PROGRAM PRG_PLAS_18_InterimCamCtrl
VAR

	bEnableInterimCameraSystem 	: BOOL;

	tofInterimCameraOFFDelay 		: TOF;

	fbInterimShiftQueue				: FB_PLAS_InterimShiftQueue;
	fbInterimCamera		: FB_SCANNER_CameraSelect;
	fbInterimEvaluation		: FB_SCANNER_Evaluation;

	rtrigNewArrived					: R_TRIG;
	bNewCodeIsProccesing			: BOOL;

	tonValidationTimout				: TON;
	bValidationTimeout				: BOOL;
	bValidationTimeoutReset			: BOOL;

	fbAddInterimCodeToQ				: FB_PLAS_AddInterimCodeToQ;
	rtrigDuplicateDetection			: R_TRIG;

	fbDebugCNT						: FB_DEBUG_CounterArray;
	aCNTDebug						: ARRAY [1..10] OF UDINT;
	bResetCNT							: BOOL;

END_VAR

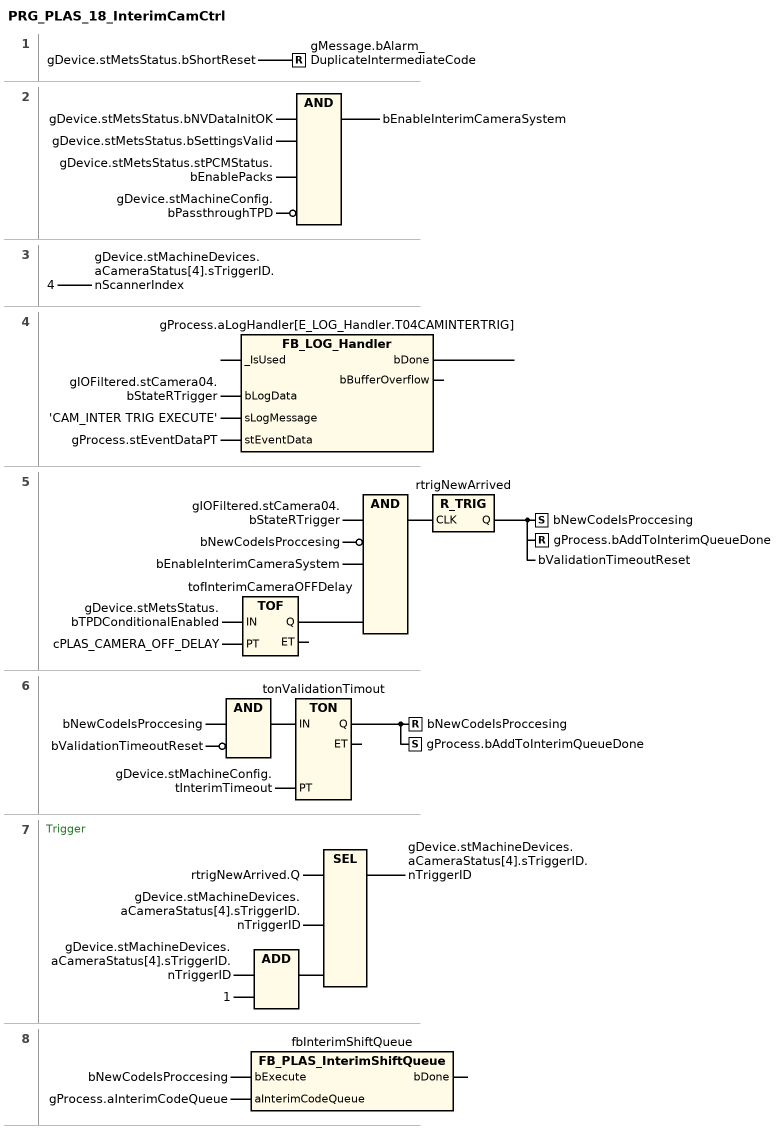
// NETWORK 1
gMessage.bAlarm_DuplicateIntermediateCode R= gDevice.stMetsStatus.bShortReset;

// NETWORK 2
bEnableInterimCameraSystem := gDevice.stMetsStatus.bNVDataInitOK AND gDevice.stMetsStatus.bSettingsValid AND gDevice.stMetsStatus.stPCMStatus.bEnablePacks AND NOT gDevice.stMachineConfig.bPassthroughTPD;

// NETWORK 3
gDevice.stMachineDevices.aCameraStatus[4].sTriggerID.nScannerIndex := 4;

// NETWORK 4
gProcess.aLogHandler[E_LOG_Handler.T04CAMINTERTRIG](
    bLogData := gIOFiltered.stCamera04.bStateRTrigger,
    sLogMessage := 'CAM_INTER TRIG EXECUTE',
    stEventData := gProcess.stEventDataPT); // FB_LOG_Handler

// NETWORK 5
tofInterimCameraOFFDelay(IN := gDevice.stMetsStatus.bTPDConditionalEnabled, PT := cPLAS_CAMERA_OFF_DELAY); // TOF
rtrigNewArrived(CLK := gIOFiltered.stCamera04.bStateRTrigger AND NOT bNewCodeIsProccesing AND bEnableInterimCameraSystem AND tofInterimCameraOFFDelay.Q); // R_TRIG
bNewCodeIsProccesing S= rtrigNewArrived.Q;
gProcess.bAddToInterimQueueDone R= rtrigNewArrived.Q;
bValidationTimeoutReset := rtrigNewArrived.Q;

// NETWORK 6
tonValidationTimout(IN := bNewCodeIsProccesing AND NOT bValidationTimeoutReset, PT := gDevice.stMachineConfig.tInterimTimeout); // TON
bNewCodeIsProccesing R= tonValidationTimout.Q;
gProcess.bAddToInterimQueueDone S= tonValidationTimout.Q;

// NETWORK 7
// Trigger
gDevice.stMachineDevices.aCameraStatus[4].sTriggerID.nTriggerID := SEL(rtrigNewArrived.Q, gDevice.stMachineDevices.aCameraStatus[4].sTriggerID.nTriggerID, gDevice.stMachineDevices.aCameraStatus[4].sTriggerID.nTriggerID + 1);

// NETWORK 8
fbInterimShiftQueue(bExecute := bNewCodeIsProccesing, aInterimCodeQueue := gProcess.aInterimCodeQueue); // FB_PLAS_InterimShiftQueue

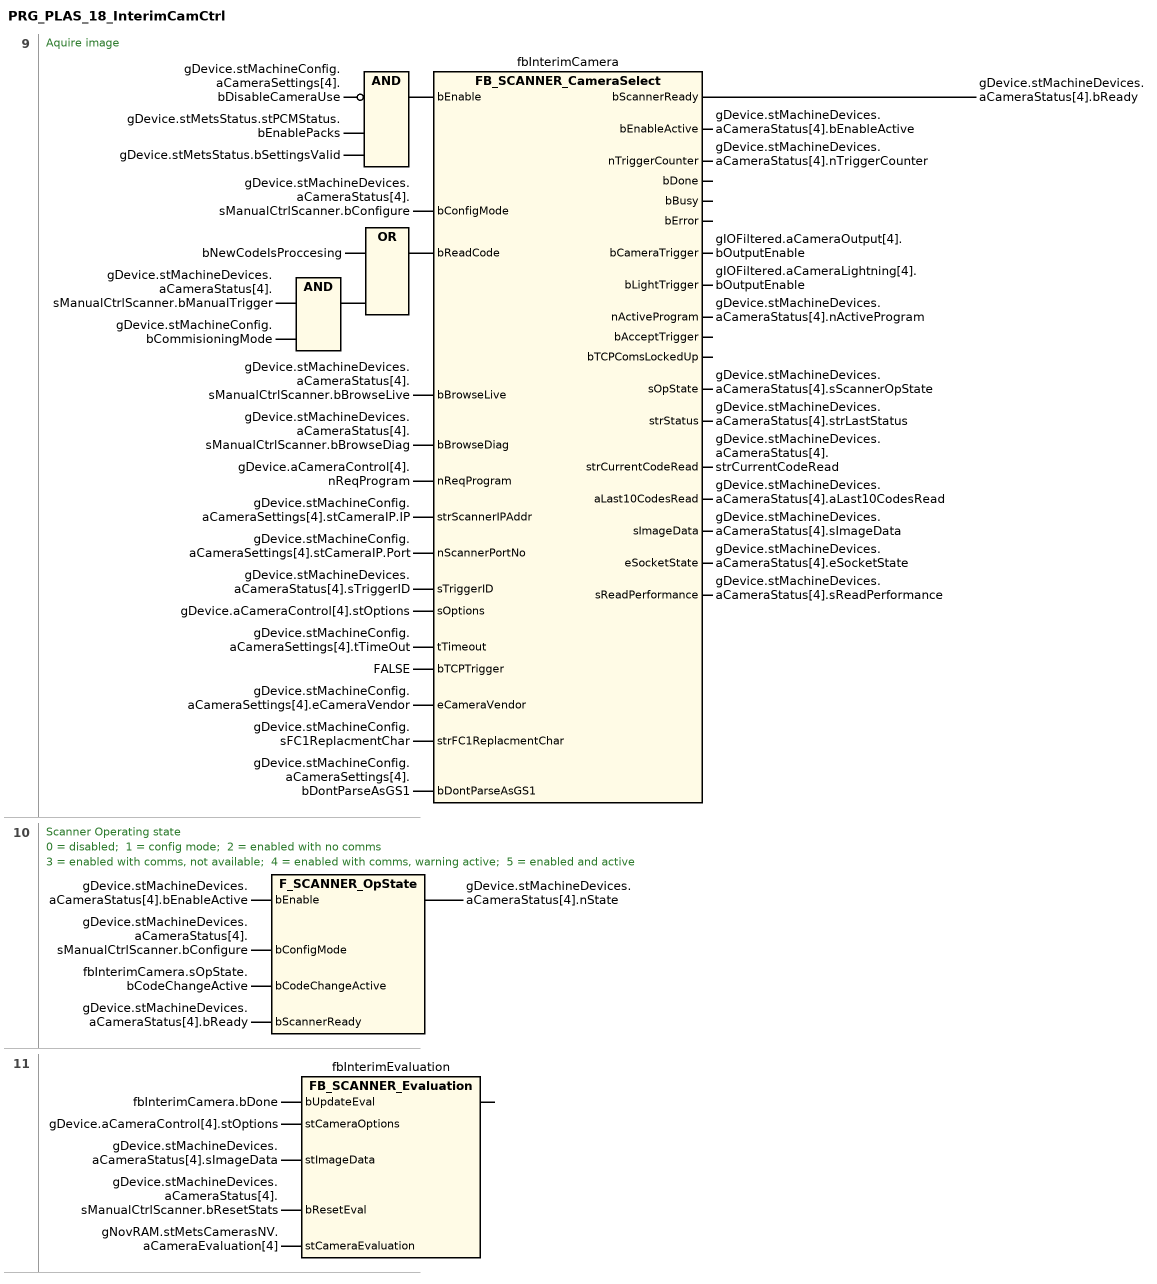
// NETWORK 9
// Aquire image
fbInterimCamera(
    bEnable := NOT gDevice.stMachineConfig.aCameraSettings[4].bDisableCameraUse AND gDevice.stMetsStatus.stPCMStatus.bEnablePacks AND gDevice.stMetsStatus.bSettingsValid,
    bConfigMode := gDevice.stMachineDevices.aCameraStatus[4].sManualCtrlScanner.bConfigure,
    bReadCode := bNewCodeIsProccesing OR gDevice.stMachineDevices.aCameraStatus[4].sManualCtrlScanner.bManualTrigger AND gDevice.stMachineConfig.bCommisioningMode,
    bBrowseLive := gDevice.stMachineDevices.aCameraStatus[4].sManualCtrlScanner.bBrowseLive,
    bBrowseDiag := gDevice.stMachineDevices.aCameraStatus[4].sManualCtrlScanner.bBrowseDiag,
    nReqProgram := gDevice.aCameraControl[4].nReqProgram,
    strScannerIPAddr := gDevice.stMachineConfig.aCameraSettings[4].stCameraIP.IP,
    nScannerPortNo := gDevice.stMachineConfig.aCameraSettings[4].stCameraIP.Port,
    sTriggerID := gDevice.stMachineDevices.aCameraStatus[4].sTriggerID,
    sOptions := gDevice.aCameraControl[4].stOptions,
    tTimeout := gDevice.stMachineConfig.aCameraSettings[4].tTimeOut,
    bTCPTrigger := FALSE,
    eCameraVendor := gDevice.stMachineConfig.aCameraSettings[4].eCameraVendor,
    strFC1ReplacmentChar := gDevice.stMachineConfig.sFC1ReplacmentChar,
    bDontParseAsGS1 := gDevice.stMachineConfig.aCameraSettings[4].bDontParseAsGS1,
    bEnableActive => gDevice.stMachineDevices.aCameraStatus[4].bEnableActive,
    nTriggerCounter => gDevice.stMachineDevices.aCameraStatus[4].nTriggerCounter,
    bCameraTrigger => gIOFiltered.aCameraOutput[4].bOutputEnable,
    bLightTrigger => gIOFiltered.aCameraLightning[4].bOutputEnable,
    nActiveProgram => gDevice.stMachineDevices.aCameraStatus[4].nActiveProgram,
    sOpState => gDevice.stMachineDevices.aCameraStatus[4].sScannerOpState,
    strStatus => gDevice.stMachineDevices.aCameraStatus[4].strLastStatus,
    strCurrentCodeRead => gDevice.stMachineDevices.aCameraStatus[4].strCurrentCodeRead,
    aLast10CodesRead => gDevice.stMachineDevices.aCameraStatus[4].aLast10CodesRead,
    sImageData => gDevice.stMachineDevices.aCameraStatus[4].sImageData,
    eSocketState => gDevice.stMachineDevices.aCameraStatus[4].eSocketState,
    sReadPerformance => gDevice.stMachineDevices.aCameraStatus[4].sReadPerformance); // FB_SCANNER_CameraSelect
gDevice.stMachineDevices.aCameraStatus[4].bReady := fbInterimCamera.bScannerReady;

// NETWORK 10
// 					Scanner Operating state
// 0 = disabled;  1 = config mode;  2 = enabled with no comms
// 3 = enabled with comms, not available;  4 = enabled with comms, warning active;  5 = enabled and active
//
gDevice.stMachineDevices.aCameraStatus[4].nState := F_SCANNER_OpState(bEnable := gDevice.stMachineDevices.aCameraStatus[4].bEnableActive, bConfigMode := gDevice.stMachineDevices.aCameraStatus[4].sManualCtrlScanner.bConfigure, bCodeChangeActive := fbInterimCamera.sOpState.bCodeChangeActive, bScannerReady := gDevice.stMachineDevices.aCameraStatus[4].bReady);

// NETWORK 11
fbInterimEvaluation(
    bUpdateEval := fbInterimCamera.bDone,
    stCameraOptions := gDevice.aCameraControl[4].stOptions,
    stImageData := gDevice.stMachineDevices.aCameraStatus[4].sImageData,
    bResetEval := gDevice.stMachineDevices.aCameraStatus[4].sManualCtrlScanner.bResetStats,
    stCameraEvaluation := gNovRAM.stMetsCamerasNV.aCameraEvaluation[4]); // FB_SCANNER_Evaluation

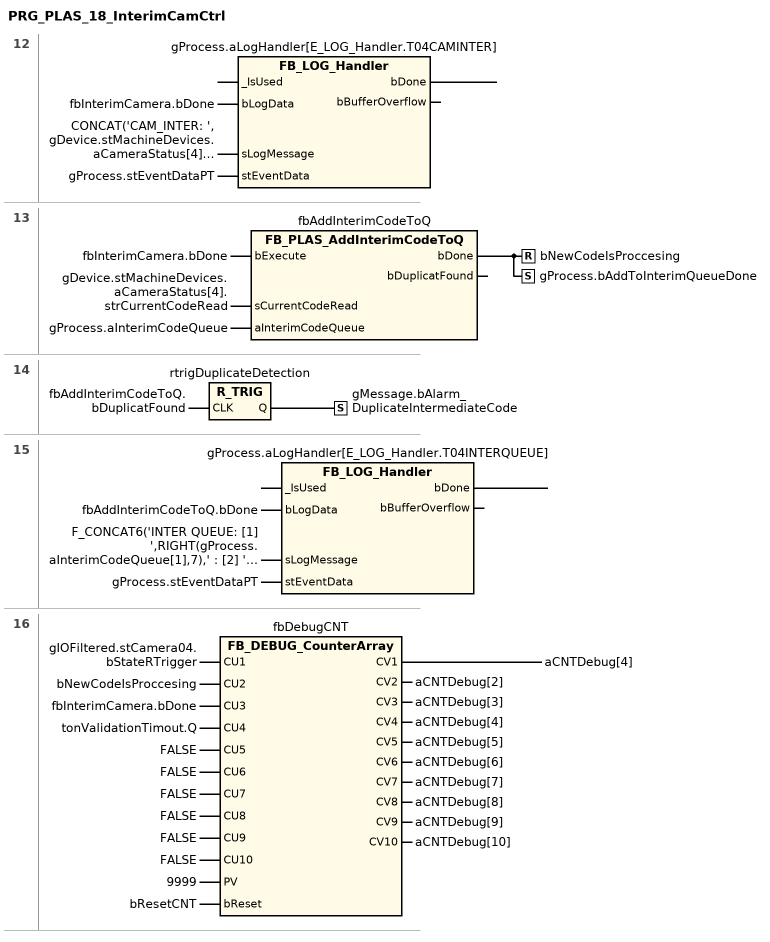
// NETWORK 12
gProcess.aLogHandler[E_LOG_Handler.T04CAMINTER](
    bLogData := fbInterimCamera.bDone,
    sLogMessage := CONCAT('CAM_INTER: ', gDevice.stMachineDevices.aCameraStatus[4].strCurrentCodeRead),
    stEventData := gProcess.stEventDataPT); // FB_LOG_Handler

// NETWORK 13
fbAddInterimCodeToQ(
    bExecute := fbInterimCamera.bDone,
    sCurrentCodeRead := gDevice.stMachineDevices.aCameraStatus[4].strCurrentCodeRead,
    aInterimCodeQueue := gProcess.aInterimCodeQueue); // FB_PLAS_AddInterimCodeToQ
bNewCodeIsProccesing R= fbAddInterimCodeToQ.bDone;
gProcess.bAddToInterimQueueDone S= fbAddInterimCodeToQ.bDone;

// NETWORK 14
rtrigDuplicateDetection(CLK := fbAddInterimCodeToQ.bDuplicatFound); // R_TRIG
gMessage.bAlarm_DuplicateIntermediateCode S= rtrigDuplicateDetection.Q;

// NETWORK 15
gProcess.aLogHandler[E_LOG_Handler.T04INTERQUEUE](
    bLogData := fbAddInterimCodeToQ.bDone,
    sLogMessage := F_CONCAT6('INTER QUEUE: [1] ',RIGHT(gProcess.aInterimCodeQueue[1],7),' : [2] ', RIGHT(gProcess.aInterimCodeQueue[2],7), ' : [3] ', RIGHT(gProcess.aInterimCodeQueue[3],7)),
    stEventData := gProcess.stEventDataPT); // FB_LOG_Handler

// NETWORK 16
fbDebugCNT(
    CU1 := gIOFiltered.stCamera04.bStateRTrigger,
    CU2 := bNewCodeIsProccesing,
    CU3 := fbInterimCamera.bDone,
    CU4 := tonValidationTimout.Q,
    CU5 := FALSE,
    CU6 := FALSE,
    CU7 := FALSE,
    CU8 := FALSE,
    CU9 := FALSE,
    CU10 := FALSE,
    PV := 9999,
    bReset := bResetCNT,
    CV2 => aCNTDebug[2],
    CV3 => aCNTDebug[3],
    CV4 => aCNTDebug[4],
    CV5 => aCNTDebug[5],
    CV6 => aCNTDebug[6],
    CV7 => aCNTDebug[7],
    CV8 => aCNTDebug[8],
    CV9 => aCNTDebug[9],
    CV10 => aCNTDebug[10]); // FB_DEBUG_CounterArray
aCNTDebug[4] := fbDebugCNT.CV1;

END_PROGRAM

(* stored: Version 1.1.0.1
   POU PRG_PLAS_18_InterimCamCtrl: Id {42f851b1-0c07-450b-b1e3-0220a31fab03}, SpecialFunc None *)
